TYPE ST_SettingsUtilities :
STRUCT
	; //To be defined
END_STRUCT
END_TYPE

(* stored: Version 1.1.0.1, ProductVersion 3.1.4024.12
   DUT ST_SettingsUtilities: Id {03c2e8fa-ccb4-4790-a1c8-8494d3221074} *)
